// TIA Portal V17 export
// export: Created 2025-06-26T06:49:12.2605615Z, ExportSetting WithDefaults, DisplayName Totally Integrated Automation Portal, DisplayVersion V17 Update 8, DisplayName TIA Portal Openness, DisplayVersion V17 Update 8, DisplayName TIA Portal Version Control Interface, DisplayVersion V17, DisplayName STEP 7 Professional, DisplayVersion V17 Update 8, DisplayName STEP 7 Safety, DisplayVersion V17 Update 6, DisplayName WinCC Advanced, DisplayVersion V17 Update 8
FUNCTION_BLOCK "PinchControl"   // FB44, FBD
TITLE = Pinch setpoint to expansion valve position
{ S7_Optimized_Access := 'TRUE' }
VERSION : 0.1
// stored: AutoNumber true, IsIECCheckEnabled false, IsRetainMemResEnabled false, MemoryReserve 40, SetENOAutomatically false, UDAEnableTagReadback false
   VAR_INPUT
      bEnable { ExternalAccessible := 'False'; ExternalVisible := 'False'; ExternalWritable := 'False'} : Bool;   // 1 = enable controller, 0 = disable controller
      bReset { ExternalAccessible := 'False'; ExternalVisible := 'False'; ExternalWritable := 'False'} : Bool;
      AddSuperheat { ExternalAccessible := 'False'; ExternalVisible := 'False'; ExternalWritable := 'False'} : Real;
   END_VAR
   VAR_OUTPUT
      EvaporationPressureLimitation { ExternalAccessible := 'False'; ExternalVisible := 'False'; ExternalWritable := 'False'} : Bool;
      CurrentPressureTarged { ExternalAccessible := 'False'; ExternalVisible := 'False'; ExternalWritable := 'False'} : Real;
   END_VAR
   VAR
      Regulator { ExternalAccessible := 'False'; ExternalVisible := 'False'; ExternalWritable := 'False'} : Struct
         x_intern_1 { ExternalAccessible := 'False'; ExternalVisible := 'False'; ExternalWritable := 'False'} : Real;
         x_intern_2 { ExternalAccessible := 'False'; ExternalVisible := 'False'; ExternalWritable := 'False'} : Real;
         x_intern_3 { ExternalAccessible := 'False'; ExternalVisible := 'False'; ExternalWritable := 'False'} : Real;
      END_STRUCT;
      AddPinch_RateOfSourceChange { ExternalAccessible := 'False'; ExternalVisible := 'False'; ExternalWritable := 'False'} : Real;
      Enabled { ExternalAccessible := 'False'; ExternalVisible := 'False'; ExternalWritable := 'False'} : Bool;
      A3030 { ExternalAccessible := 'False'; ExternalVisible := 'False'; ExternalWritable := 'False'} : "fbHMIEvent";
   END_VAR
   VAR_TEMP
      PIDControlInactive : Bool;   // if true set "#StaticOutputValue" to expansionvalves
      StaticOutputValue : Real;   // setpoint for expansionfalves if not "PIDControlInactive"
   END_VAR
   VAR CONSTANT
      EXP_VLV_PID_CALMING : Real := 27.0;   // Super Heat Temperature that reduces Control Ampfication by 64%
   END_VAR
BEGIN

REGION Network 1: Reset manual mode
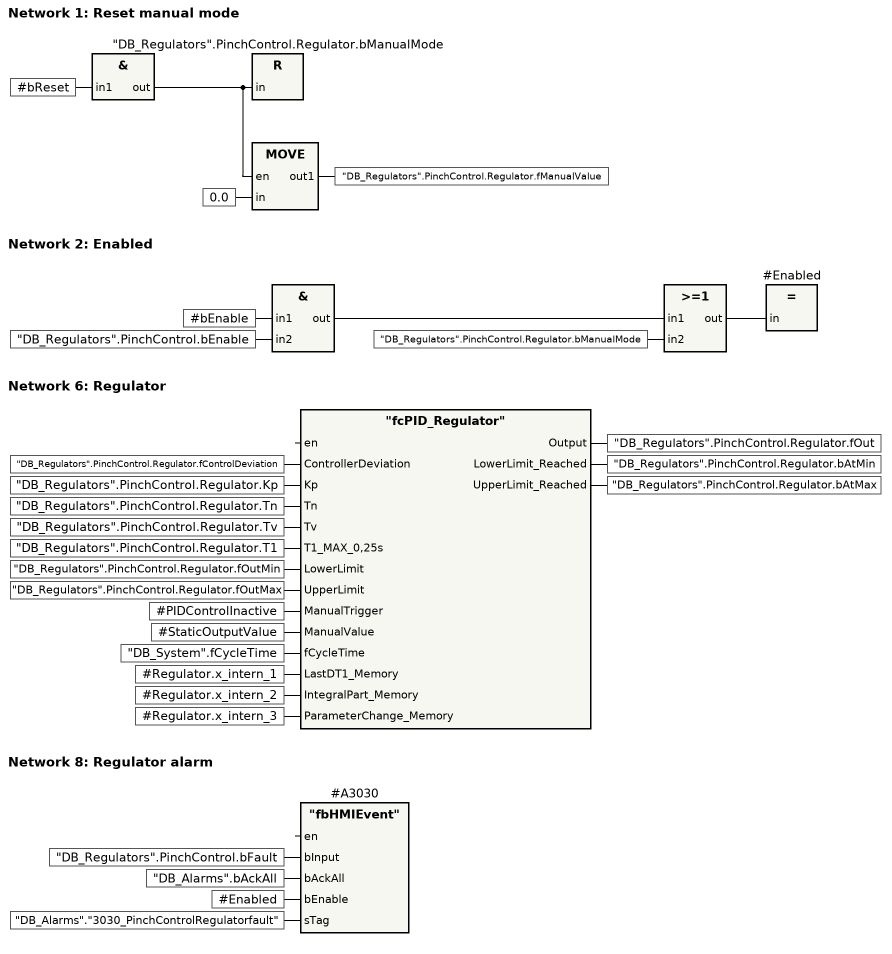
   IF #bReset THEN
       "DB_Regulators".PinchControl.Regulator.bManualMode := FALSE;
       "DB_Regulators".PinchControl.Regulator.fManualValue := 0.0;
   END_IF;
END_REGION

REGION Network 2: Enabled
   #Enabled := (#bEnable AND "DB_Regulators".PinchControl.bEnable) OR "DB_Regulators".PinchControl.Regulator.bManualMode;
END_REGION

REGION Network 3 (SCL): Static output
   // ###CHANGE: Added complete network:
   // If the controller is inactive and the expansion valve and the controller is set to an fixed value.
   IF ("DB_Regulators".PinchControl.Regulator.bManualMode) THEN
       // Set expansion valve to manual setpoint
       #StaticOutputValue := "DB_Regulators".PinchControl.Regulator.fManualValue;
   ELSIF ("DB_State".State."4_Start") THEN
       //Set expansion valves to fixed opening on startup
       //###CHANGE: The function to close the expansion valve if the compressor is stopped in dryout.
       //###CHANGE: Added the flag "DB_Regulators".PurgeControl.bDone = 0 since in state 4, in dyout (after purge), the "DB_Regulators".PurgeControl.bSpinning is zero but the comperssor is turning again. 
       IF ("DB_Regulators".PurgeControl.bSpinning = 0 AND "DB_Regulators".PurgeControl.bDone = 0) THEN
           #StaticOutputValue := 0;
       //###CHANGE: New function TO limit massflow on dryout with already filled evaporator at evaporation pressure > 300kPa.    
       ELSIF ("DB_AI".HBL_PT_572.Eng.fValue > 300.0) THEN   // 300kPa is larger than dryout pressure and sat at ~minimalinlet temperature. // 300kPa should be auto calculated or part of the dataset
           //###Note: With more than 300kPa we can assume that the evaporator is still filled and an additional amount of refrigerant would not be helpful
           #StaticOutputValue := "DB_CurrentSetting".MissingSetting.System.ExpansionValvePositionStartCold;
       ELSE
           #StaticOutputValue := "DB_CurrentSetting".MissingSetting.System.ExpansionValvePositionStart;
       END_IF;
   ELSIF (NOT #Enabled) THEN
       // Close expansion valve if inactive
       #StaticOutputValue := 0;
   END_IF;

   //Inactivate PID controler if a upper condition is fulfilled. Controler is reset to current output if true
   #PIDControlInactive := NOT #Enabled OR "DB_State".State."4_Start"OR"DB_Regulators".PinchControl.Regulator.bManualMode;
END_REGION

REGION Network 4 (SCL): Pinch setpoint
   // Setpoint is the pinch from the superheat regulator
   "DB_Regulators".PinchControl.fSetpoint := "DB_Regulators".SuperheatControl.Regulator.fOut;

   // Additional superheat
   "DB_Regulators".PinchControl.fSetpoint += 0.35 * #AddSuperheat * LIMIT_REAL(IN := "DB_Regulators".PinchControl.fSetpoint /"DB_Calc".LowPressPart.CompressorSuperheat.fValue, MN := 0,MX:=1); // Pilot-control-filter to bypass additional superheat to the pinch controller

   // Preliminary setpoint modification to counteract source temperature changes
   #AddPinch_RateOfSourceChange := -3.0 * "DB_Calc".HeatSource.TemperatureRateOfChange.fValue;

   IF #AddPinch_RateOfSourceChange > -0.75 * "DB_Regulators".PinchControl.fSetpoint THEN //Maximum compensation is 75% of unmodified Setpoint
       "DB_Regulators".PinchControl.fSetpoint += #AddPinch_RateOfSourceChange;
   ELSE
       //The internal value of the DT1-Block is also corrected by the leftover to enable a rapid response in case of a change of direction.
       (*#DT1_Merker_intern -= #AddPinch_RateOfSourceChange + 0.75 * #DB_Regulators.ExpansionValve.fSetpoint;*)
       //To avoid overcorrection the temperature change correction is limited to the left 25%.
       "DB_Regulators".PinchControl.fSetpoint *= 0.25;
   END_IF;
END_REGION

REGION Network 5 (SCL): Deviation
   //The control error is the difference between current pinch value and pinch setpoint.
   IF ("DB_Calc".HeatSource.Pinch.bError = TRUE) OR "isNaN"("DB_Regulators".PinchControl.fSetpoint) OR ("DB_Calc".Misc.EvaporatorDischargePressureMean.bError = TRUE) THEN
       "DB_Regulators".PinchControl.Regulator.fControlDeviation := 0;
       "DB_Regulators".PinchControl.bFault := TRUE;
   ELSE
       "DB_Regulators".PinchControl.bFault := FALSE;
       "DB_Regulators".PinchControl.Regulator.fControlDeviation := "DB_Calc".HeatSource.Pinch.fValue - "DB_Regulators".PinchControl.fSetpoint;

       // Maximum suction pressure protection
       // The target evaporation temperature should ensure a boiling pressure of no more than 1000 kPa (Maximum Limit - 100kPa). For this purpose, the control error is limited in case of a high evaporation pressure/temperature.
       IF "DB_Regulators".PinchControl.Regulator.fControlDeviation > (("DB_CurrentSetting".Compressor.Limits.p_CrankCase_Max - 100.0) - "DB_Calc".Misc.EvaporatorDischargePressureMean.fValue) THEN
           "DB_Regulators".PinchControl.Regulator.fControlDeviation := (("DB_CurrentSetting".Compressor.Limits.p_CrankCase_Max - 100.0) - "DB_Calc".Misc.EvaporatorDischargePressureMean.fValue) / 10.0;
           #EvaporationPressureLimitation := True;
       ELSE
           #EvaporationPressureLimitation := False;
       END_IF;

       // Current pressure target for visualisation and debugging
       #CurrentPressureTarged := "DB_Regulators".PinchControl.Regulator.fControlDeviation + "DB_Calc".Misc.EvaporatorDischargePressureMean.fValue;

       //Adapt Pinch control Kp-factor:
       //We need this function because an unloaded ("empty") evaporator reacts very sensitively to a changed refrigerant quantity. Empty or unloaded always means relatively much superheat, so that we can fine-tune it with this value.
       //The Kp factor depends on the Superheat after the Evaporator. If there is much superheat, the kp is smaller and if the superheat gets to zero it gets closer to the preset factor (3.0). A superheat of #EXP_VLV_PID_CALMING (14K) reduces Kp by 64% and a superheat of 2*#EXP_VLV_PID_CALMING reduces the Kp by 86%.
       "DB_Regulators".PinchControl.Regulator.Kp := 0.8 * LIMIT_REAL(IN := EXP((0.5 * "DB_Regulators".PinchControl.Regulator.fControlDeviation - "DB_Calc".LowPressPart.EvaporatorSuperheat.fValue) / #EXP_VLV_PID_CALMING), MN := 0.1, MX := 1);

       // The Lower limit for the expansion valve position can be increased on warmup
       // To ensure a minimal "heat" flow a minimal leakage might be helpful 
       IF "DB_State".State."5_Warmup" THEN
           "DB_Regulators".PinchControl.Regulator.fOutMin := "DB_CurrentSetting".MissingSetting.System.ExpansionValvePositionStart;
       ELSE
           "DB_Regulators".PinchControl.Regulator.fOutMin := 2.5;
       END_IF;
   END_IF;
END_REGION

REGION Network 6: Regulator
   "fcPID_Regulator"(ControllerDeviation := "DB_Regulators".PinchControl.Regulator.fControlDeviation,
                     Kp := "DB_Regulators".PinchControl.Regulator.Kp,
                     Tn := "DB_Regulators".PinchControl.Regulator.Tn,
                     Tv := "DB_Regulators".PinchControl.Regulator.Tv,
                     "T1_MAX_0,25s" := "DB_Regulators".PinchControl.Regulator.T1,
                     LowerLimit := "DB_Regulators".PinchControl.Regulator.fOutMin,
                     UpperLimit := "DB_Regulators".PinchControl.Regulator.fOutMax,
                     ManualTrigger := #PIDControlInactive,
                     ManualValue := #StaticOutputValue,
                     fCycleTime := "DB_System".fCycleTime,
                     LastDT1_Memory := #Regulator.x_intern_1,
                     IntegralPart_Memory := #Regulator.x_intern_2,
                     ParameterChange_Memory := #Regulator.x_intern_3,
                     Output => "DB_Regulators".PinchControl.Regulator.fOut,
                     LowerLimit_Reached => "DB_Regulators".PinchControl.Regulator.bAtMin,
                     UpperLimit_Reached => "DB_Regulators".PinchControl.Regulator.bAtMax);
END_REGION

REGION Network 7 (SCL): Disable
   IF #PIDControlInactive = True THEN
       "DB_Regulators".PinchControl.Regulator.fOut := #StaticOutputValue;
       "DB_Regulators".PinchControl.Regulator.bAtMin := FALSE;
       "DB_Regulators".PinchControl.Regulator.bAtMax := FALSE;
   END_IF;
END_REGION

REGION Network 8: Regulator alarm
   #A3030(bInput := "DB_Regulators".PinchControl.bFault,   // "fbHMIEvent"
          bAckAll := "DB_Alarms".bAckAll,
          bEnable := #Enabled,
          sTag := "DB_Alarms"."3030_PinchControlRegulatorfault");
END_REGION

REGION Network 9 (SCL): Mode
   // Mode
   IF "DB_Regulators".PinchControl.Regulator.bManualMode = TRUE THEN
       "DB_Regulators".PinchControl.nMode := 2;
   ELSIF "DB_Regulators".PinchControl.bEnable = TRUE THEN
       "DB_Regulators".PinchControl.nMode := 1;
   ELSE
       "DB_Regulators".PinchControl.nMode := 0;
   END_IF;
END_REGION
END_FUNCTION_BLOCK
